Yaskawa INFORM job: INITIALISATION.JBI

/JOB
//NAME INITIALISATION
//POS
///NPOS 0,0,0,0,0,0
//INST
///DATE 2018/09/03 15:31
///ATTR SC,RW
NOP
'*****
'initialisation
DOUT OG#(68) 0
DOUT OG#(69) 0
DOUT OG#(70) 0
DOUT OG#(71) 0
DOUT OG#(74) 0
DOUT OG#(75) 0
DOUT OG#(76) 0
DOUT OG#(77) 0
DOUT OG#(78) 0
DOUT OG#(79) 0
END
